// TIA Portal V19 export
FUNCTION_BLOCK "SCALE"   // FB1, LAD
{ S7_Optimized_Access := 'TRUE' }
// stored: MemoryReserve 100, SetENOAutomatically false
   VAR_INPUT
      "SCALE MIN" : Real;
      "SCALE MAX" : Real;
      INPUT : Int;
      RAW_MIN : Int;
      RAW_MAX : Int;
   END_VAR
   VAR_OUTPUT
      PV_VALUE : Real;
   END_VAR
   VAR_IN_OUT
      NORM_X : Real;
   END_VAR
BEGIN

REGION Network 1
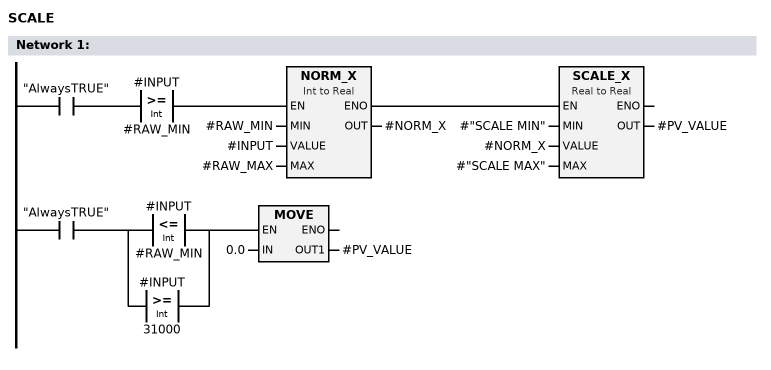
   RUNG wire#powerrail
      Contact( "AlwaysTRUE" )
      { S7_Templates := "SrcType := Int" } GE_Contact(in1 := #INPUT, in2 := #RAW_MIN)
      { S7_Templates := "[SrcType := Int, DestType := Real]" } Normalize(min := #RAW_MIN, value := #INPUT, max := #RAW_MAX, out => #NORM_X)
      { S7_Templates := "[SrcType := Real, DestType := Real]" } Scale(min := #"SCALE MIN", value := #NORM_X, max := #"SCALE MAX", out => #PV_VALUE)
   END_RUNG
   RUNG wire#powerrail
      Contact( "AlwaysTRUE" )
      wire#w1
      { S7_Templates := "SrcType := Int" } LE_Contact(in1 := #INPUT, in2 := #RAW_MIN)
      wire#w2
      Move(in := 0.0, out1 => #PV_VALUE)
   END_RUNG
   RUNG wire#w1
      { S7_Templates := "SrcType := Int" } GE_Contact(in1 := #INPUT, in2 := 31000)
   END_RUNG wire#w2
   // the same network as SCL:
   IF "AlwaysTRUE" AND (#INPUT >= #RAW_MIN) THEN
       #NORM_X := NORM_X(MIN := #RAW_MIN, VALUE := #INPUT, MAX := #RAW_MAX);
       #PV_VALUE := SCALE_X(MIN := #"SCALE MIN", VALUE := #NORM_X, MAX := #"SCALE MAX");
   END_IF;
   IF "AlwaysTRUE" AND ((#INPUT <= #RAW_MIN) OR (#INPUT >= 31000)) THEN #PV_VALUE := 0.0; END_IF;
END_REGION
END_FUNCTION_BLOCK
